// Interlock logic for the Amphos shutter
FUNCTION F_AmphosShutterEnable : BOOL
VAR_INPUT
    //bAmphosOn : BOOL; // Whether the amphos is on
    fOpcpaVoltage           : LREAL; // The voltage of the OPCPA
    fAmphosVoltage          : LREAL; // The Amphos voltage
    AmphosStatus            : BOOL; //Amphos Laser Shutter Status
    bLoopTempOverride01     : BOOL; // Whether the chiller loop error is overriden
    bLoopTempOverride02     : BOOL; // Whether the chiller loop error is overriden
    bLoopTempOverride03     : BOOL; // Whether the chiller loop error is overriden
    bLoopTempOverride04     : BOOL; // Whether the chiller loop error is overriden
    bLoopTempOverride05     : BOOL; // Whether the chiller loop error is overriden
    ShutterStatus : BOOL; //Shutter Status
END_VAR

VAR_IN_OUT CONSTANT
    stErrors                : ST_ErrorStates; // Currently detected errors
    stOpcpaSetpoints        : ST_LaserSetpoints; // OPCPA setpoints
    stAmphosSetpoints       : ST_LaserSetpoints; // The Amphos setpoints
    Mode                    : E_Mode; // Mode of operation
END_VAR

VAR
    bAmphosUnderVolt        : BOOL; // Amphos Power meter under min setpoint voltage
    bOpcpaUnderVolt         : BOOL; // OPCPA Power meter under min setpoint voltage
    bChillerErrors          : BOOL; // Any chiller loop errors but is not manually overridden
    bOverTempErrors         : BOOL; // Any temperature switch errors
END_VAR

(*// The Amphos Shutter Enable function sends and Enable or Disable bit as an output to be used by the Amphos Shutter Command block
// AmphosShutterEnable := True := OPEN SHUTTER
// AmphosShutterEnable := FALSE := CLOSE SHUTTER
The below logic follows the logic table
Note : In master override modes, the Shutter state will hold the previous state value, unless manually forced
*)
// consolidate the check for temperature overrides and chiller loop errors
bChillerErrors := (
                   (NOT bLoopTempOverride01 AND stErrors.bChillerLoop01) OR
                   (NOT bLoopTempOverride02 AND stErrors.bChillerLoop02) OR
                   (NOT bLoopTempOverride03 AND stErrors.bChillerLoop03) OR
                   (NOT bLoopTempOverride04 AND stErrors.bChillerLoop04)OR
                   (NOT bLoopTempOverride05 AND stErrors.bChillerLoop05)
                   );
// consolidate temperature switch faults. Remember, they are NC, so FALSE means ERROR
bOverTempErrors := (NOT GVL_IO.bLoopTempSW01 OR
                    NOT GVL_IO.bLoopTempSW02 OR
                    NOT GVL_IO.bLoopTempSW03 OR
                    NOT GVL_IO.bLoopTempSW04 OR
                    NOT GVL_IO.bLoopTempSW05);

bAmphosUnderVolt := fAmphosVoltage < stAmphosSetpoints.nMinVoltage;
bOpcpaUnderVolt := fOpcpaVoltage < stOpcpaSetpoints.nMinVoltage;

// Close shutter if there is a hardware failure
IF stErrors.bHardwareFailure
   // Close shutter if there is a leak on the optical table with the amphos on, a leak under the table, or a leak inside the OPCPA with Carbide on
   // OR stErrors.bLeakOpticalTableAmphosOn OR stErrors.bLeakOpcpaCarbideOn OR stErrors.bLeakUnderTable
    OR (bChillerErrors or bOverTempErrors)
    // Close shutter if in OPCPA beam error state and OPCPA voltage too low
    OR (bOpcpaUnderVolt AND stErrors.bOpcpaBeam)
    // Close shutter if there is a Dump Chiller error
    OR stErrors.bDumpChiller
    OR (NOT GVL_IO.bDumpChillerFlow)
    OR (NOT GVL_IO.bBaseplateChillerFlow)
THEN
    F_AmphosShutterEnable := FALSE;
ELSE
    CASE MODE OF
        E_Mode.MASTER_Override, E_Mode.Maintenance:
            IF NOT ShutterStatus
            THEN
                F_AmphosShutterEnable := TRUE;
            ELSE
                F_AmphosShutterEnable := FALSE;
            END_IF
        E_Mode.Protection:
            IF bAmphosUnderVolt OR bOpcpaUnderVolt OR NOT AmphosStatus
            THEN
                F_AmphosShutterEnable := FALSE;
            ELSE
                F_AmphosShutterEnable := TRUE;
            END_IF
        // Undefined state, do not get here
        ELSE
            Mode := E_Mode.Protection;
    END_CASE
END_IF

END_FUNCTION

(* stored: Version 1.1.0.1, ProductVersion 3.1.4024.12
   POU F_AmphosShutterEnable: Id {a7fc5b7f-48ee-48e8-a6f9-0fc0af7200c2}, SpecialFunc None *)
